(* IEC 61131-3 sources: volt/packages/volt-lsp-iec/test-corpus/pro2193/Device/Plc Logic/Application/09 Misc/Library Manager/BreakpointLogging, 3 files *)

(* ---- VARIABLES.gvl ---- *)
VAR_GLOBAL
	STLOGSTRING : STRING(255);
	PLOGSTRING : POINTER TO STRING(255) := ADR(stLogString);
END_VAR

(* ---- APPENDTOSTRING.pou ---- *)
FUNCTION APPENDTOSTRING : BOOL
VAR_INPUT
	HEAD : POINTER TO STRING(255);
	TAIL : STRING(255);
END_VAR
END_FUNCTION

(* ---- LOGTODEVICE.pou ---- *)
FUNCTION LOGTODEVICE : BOOL
VAR_INPUT
	PMESSAGE : POINTER TO STRING(255);
END_VAR
END_FUNCTION
